SYSTEM SFP-Server
  (* Version 1.0, Author, 4DIAC-Consortium *)
  APPLICATION singleTag
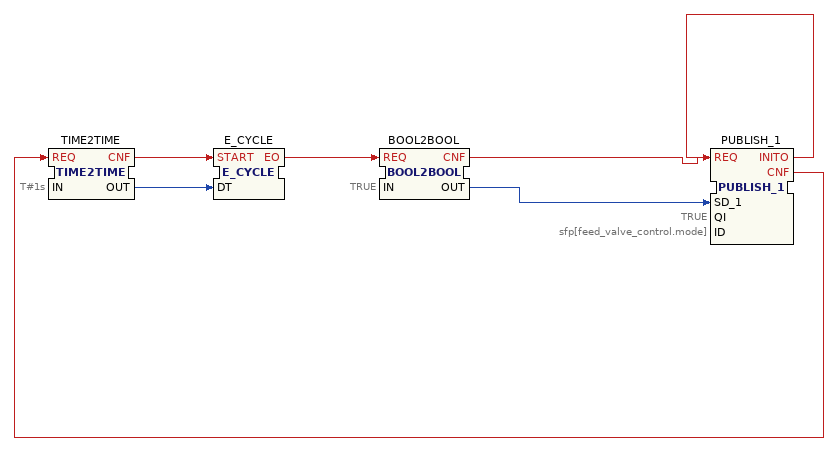
    FBS
      BOOL2BOOL : BOOL2BOOL(IN := TRUE);
      PUBLISH_1 : PUBLISH_1(QI := TRUE, ID := sfp[feed_valve_control.mode]);
      E_CYCLE : E_CYCLE;
      TIME2TIME : TIME2TIME(IN := T#1s);
    END_FBS
    EVENT_CONNECTIONS
      E_CYCLE.EO TO BOOL2BOOL.REQ;
      PUBLISH_1.INITO TO PUBLISH_1.REQ;
      BOOL2BOOL.CNF TO PUBLISH_1.REQ;
      PUBLISH_1.CNF TO TIME2TIME.REQ;
      TIME2TIME.CNF TO E_CYCLE.START;
    END_CONNECTIONS
    DATA_CONNECTIONS
      BOOL2BOOL.OUT TO PUBLISH_1.SD_1;
      TIME2TIME.OUT TO E_CYCLE.DT;
    END_CONNECTIONS
  END_APPLICATION
  APPLICATION tesreconf
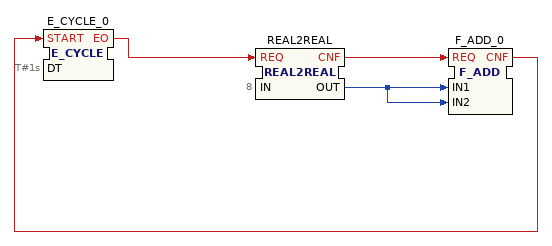
    FBS
      E_CYCLE_0 : E_CYCLE(DT := T#1s);
      REAL2REAL : REAL2REAL(IN := 8);
      F_ADD_0 : F_ADD;
    END_FBS
    EVENT_CONNECTIONS
      E_CYCLE_0.EO TO REAL2REAL.REQ;
      REAL2REAL.CNF TO F_ADD_0.REQ;
      F_ADD_0.CNF TO E_CYCLE_0.START;
    END_CONNECTIONS
    DATA_CONNECTIONS
      REAL2REAL.OUT TO F_ADD_0.IN1;
      REAL2REAL.OUT TO F_ADD_0.IN2;
    END_CONNECTIONS
  END_APPLICATION
  APPLICATION test_new
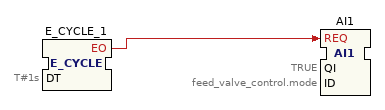
    FBS
      AI1 : AI1(QI := TRUE, ID := feed_valve_control.mode);
      E_CYCLE_1 : E_CYCLE(DT := T#1s);
    END_FBS
    EVENT_CONNECTIONS
      E_CYCLE_1.EO TO AI1.REQ;
    END_CONNECTIONS
  END_APPLICATION
  DEVICE FORTE_PC : FORTE_PC(MGR_ID := "localhost:61499")
    {SET_ATTRIBUTE(Profile, HOLOBLOC)}
    RESOURCE EMB_RES : EMB_RES
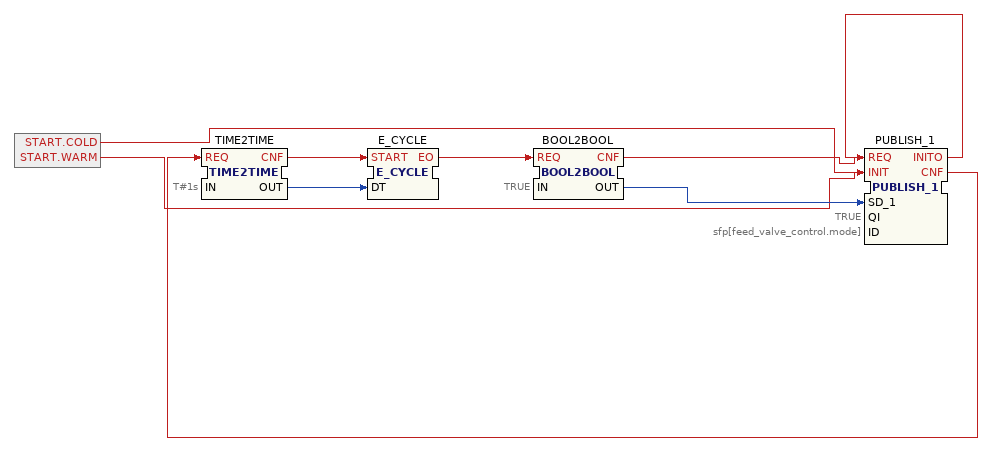
      FBS
        BOOL2BOOL : BOOL2BOOL(IN := TRUE);
        PUBLISH_1 : PUBLISH_1(QI := TRUE, ID := sfp[feed_valve_control.mode]);
        E_CYCLE : E_CYCLE;
        TIME2TIME : TIME2TIME(IN := T#1s);
      END_FBS
      EVENT_CONNECTIONS
        PUBLISH_1.INITO TO PUBLISH_1.REQ;
        BOOL2BOOL.CNF TO PUBLISH_1.REQ;
        E_CYCLE.EO TO BOOL2BOOL.REQ;
        PUBLISH_1.CNF TO TIME2TIME.REQ;
        TIME2TIME.CNF TO E_CYCLE.START;
        START.COLD TO PUBLISH_1.INIT;
        START.WARM TO PUBLISH_1.INIT;
      END_CONNECTIONS
      DATA_CONNECTIONS
        BOOL2BOOL.OUT TO PUBLISH_1.SD_1;
        TIME2TIME.OUT TO E_CYCLE.DT;
      END_CONNECTIONS
    END_RESOURCE
  END_DEVICE
  MAPPINGS
    singleTag.BOOL2BOOL ON FORTE_PC.EMB_RES.BOOL2BOOL;
    singleTag.PUBLISH_1 ON FORTE_PC.EMB_RES.PUBLISH_1;
    singleTag.E_CYCLE ON FORTE_PC.EMB_RES.E_CYCLE;
    singleTag.TIME2TIME ON FORTE_PC.EMB_RES.TIME2TIME;
  END_MAPPINGS
  SEGMENTS
    Ethernet : Ethernet;
  END_SEGMENTS
  LINKS
    FORTE_PC => Ethernet;
  END_LINKS
END_SYSTEM
